FUNCTION_BLOCK POU_extend EXTENDS AxisBase
VAR_INPUT
END_VAR
VAR_OUTPUT
END_VAR
VAR
	fbReadMotorTemp: FB_SoEReadMotorTemperature;
END_VAR

fbReadMotorTemp(
	Axis :=axis,
	NetId := ,
	Execute := ,
	Timeout := ,
	Busy => ,
	Error => ,
	AdsErrId => ,
	SercosErrId => ,
	MotorTemperature =>,
	Attribute => );

END_FUNCTION_BLOCK

(* stored: Version 1.1.0.1, ProductVersion 3.1.4024.12
   POU POU_extend: Id {9c3bf9c5-ce22-4e23-b99d-fa297be233f2}, SpecialFunc None *)
